(* IEC 61131-3 sources: Industry-PLC-LLM/data/PLCBEAD_repo/PLCBEAD_PLCEmbed-main/PLC-BEAD/Source/GEB/STACK_16, 1 file *)

(* ---- STACK_16.ST ---- *)
TYPE
  oscat_ardw_0_15             : ARRAY [0..15]   OF DWORD;
END_TYPE

FUNCTION_BLOCK STACK_16_Block

	VAR_INPUT
		DIN :	DWORD;
		E :	BOOL := TRUE;
		RD :	BOOL;
		WD :	BOOL;
		RST :	BOOL;
	END_VAR

	VAR_OUTPUT
		DOUT :	DWORD;
		EMPTY :	BOOL := TRUE;
		FULL :	BOOL;
	END_VAR

	VAR
		PT :	INT;
		stack :	oscat_ardw_0_15;
	END_VAR

	IF RST THEN
		PT := 0;
		EMPTY := TRUE;
		FULL := FALSE;
		DOUT := DWORD#0;
	ELSIF E THEN
		IF NOT EMPTY AND RD THEN
			PT := PT - 1;
			DOUT := stack[PT];
			EMPTY := PT = 0;
			FULL := FALSE;
		END_IF;
		IF NOT FULL AND WD THEN
			stack[PT] := Din;
			PT := PT + 1;
			FULL := PT > 15;
			EMPTY := FALSE;
		END_IF;
	END_IF;

END_FUNCTION_BLOCK

PROGRAM program0
	VAR
		DIN :	DWORD;
		E :	BOOL := TRUE;
		RD :	BOOL;
		WD :	BOOL;
		RST :	BOOL;
		DOUT :	DWORD;
		EMPTY :	BOOL := TRUE;
		FULL :	BOOL;
		func_block : STACK_16_Block;
	END_VAR
		func_block.DIN  := DIN;
		func_block.E  := E;
		func_block.RD  := RD;
		func_block.WD  := WD;
		func_block.RST  := RST;
		func_block();
		DOUT := func_block.DOUT;
		EMPTY := func_block.EMPTY;
		FULL := func_block.FULL;

END_PROGRAM
